// TIA Portal V20 export
TYPE "PartStatus2"
// stored: Access Published
   STRUCT
      Reserved_0 : Bool;
      Reserved_1 : Bool;
      Reserved_2 : Bool;
      Reserved_3 : Bool;
      Reserved_4 : Bool;
      Reserved_5 : Bool;
      Reserved_6 : Bool;
      Reserved_7 : Bool;
   END_STRUCT;
END_TYPE
